// TIA Portal V17 export
// export: Created 2023-12-22T15:28:29.4431312Z, ExportSetting WithDefaults, DisplayName Totally Integrated Automation Portal, DisplayVersion V17, DisplayName TIA Portal Openness, DisplayVersion V17, DisplayName TIA Portal Version Control Interface, DisplayVersion V17, DisplayName STEP 7 Professional, DisplayVersion V17, DisplayName STEP 7 Safety, DisplayVersion V17, DisplayName WinCC Advanced, DisplayVersion V17
FUNCTION_BLOCK "Time_H"   // FB93, LAD
{ S7_Optimized_Access := 'FALSE' }
VERSION : 0.1
// stored: AutoNumber false, IsIECCheckEnabled false, SetENOAutomatically false, UDAEnableTagReadback false
   VAR DB_SPECIFIC
      SP_H { S7_SetPoint := 'True'} : DInt;   // Уставка часов - от 0 до 999
      SP_M { S7_SetPoint := 'True'} : DInt;   // Уставка минут - от 0 до 59
      SP_S { S7_SetPoint := 'True'} : DInt;   // Уставка секунд - от 0 до 59
      Now_H : DInt;   // Прошло часов от начала отсчёта
      Now_M : DInt;   // Прошло минут от начала отсчёта
      Now_S : DInt;   // Прошло секунд от начала отсчёта
      Rev_H : DInt;   // Осталось часов до уставки
      Rev_M : DInt;   // Осталось минут до уставки
      Rev_S : DInt;   // Осталось секунд до уставки
      Progress : Real;   // Прогресс выполнения
      Start : Bool;   // Запуск
      "Exit" : Bool;   // Счёт завершён
      Pause : Bool;   // Пауза
      Reset : Bool;   // Сброс таймера
   END_VAR
   VAR_TEMP
      Full_SP_S : DInt;
      Full_Now_S : DInt;
      Full_Delta_S : DInt;
      x1 : DInt;
      x2 : DInt;
   END_VAR
   VAR_TEMP   // added for the SCL form of the ladder/FBD networks
      _w1 : Bool;
      _w2 : Bool;
   END_VAR
BEGIN

REGION Network 1: Подсчёт времени
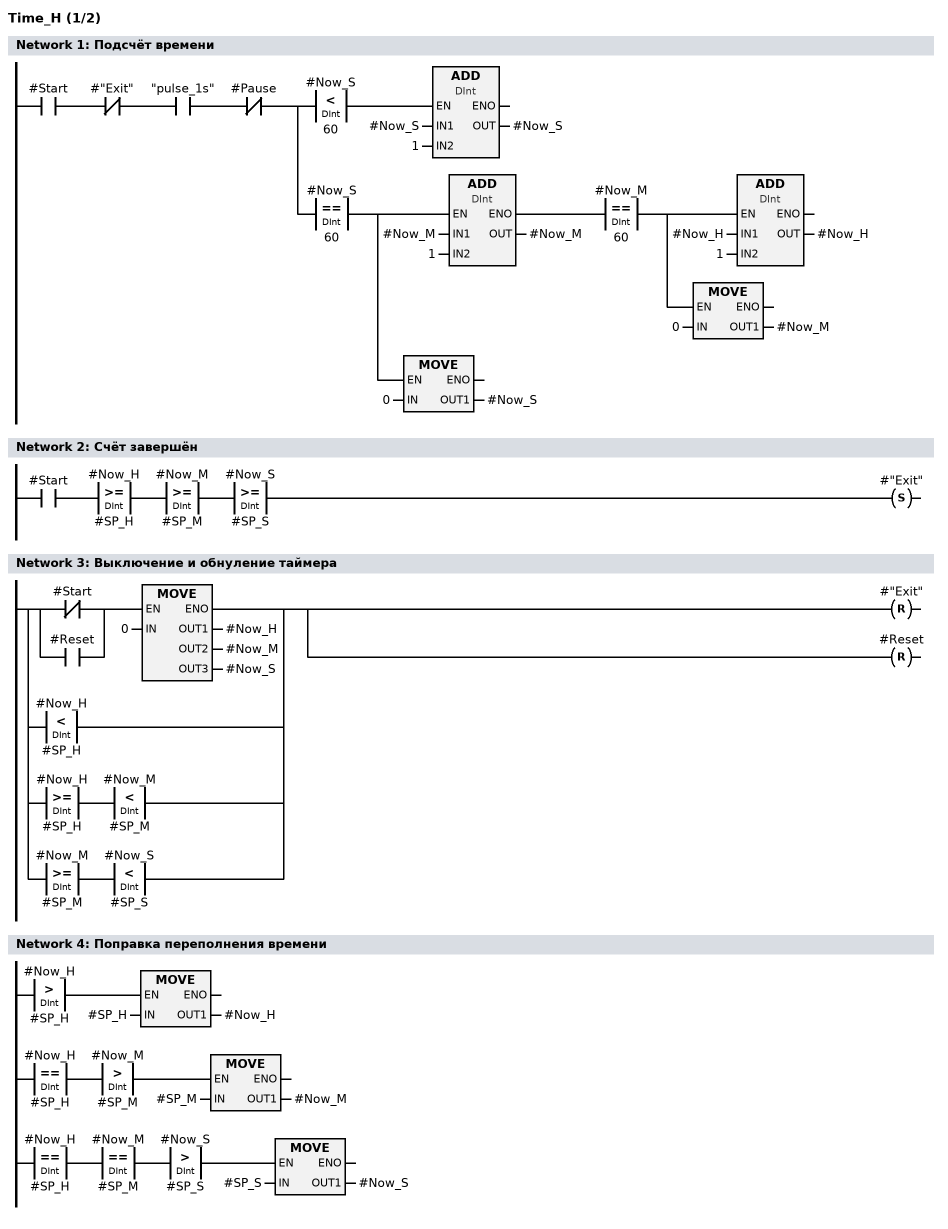
   RUNG wire#powerrail
      Contact( #Start )
      I_Contact( #"Exit" )
      Contact( "pulse_1s" )
      I_Contact( #Pause )
      wire#w1
      { S7_Templates := "SrcType := DInt" } LT_Contact(in1 := #Now_S, in2 := 60)
      { S7_Templates := "SrcType := DInt"; S7_GenerateENO := "TRUE" } Add(in1 := #Now_S, in2 := 1, out => #Now_S)
   END_RUNG
   RUNG wire#w1
      { S7_Templates := "SrcType := DInt" } EQ_Contact(in1 := #Now_S, in2 := 60)
      wire#w2
      { S7_Templates := "SrcType := DInt"; S7_GenerateENO := "TRUE" } Add(in1 := #Now_M, in2 := 1, out => #Now_M)
      { S7_Templates := "SrcType := DInt" } EQ_Contact(in1 := #Now_M, in2 := 60)
      wire#w3
      { S7_Templates := "SrcType := DInt"; S7_GenerateENO := "TRUE" } Add(in1 := #Now_H, in2 := 1, out => #Now_H)
   END_RUNG
   RUNG wire#w3
      { S7_GenerateENO := "TRUE" } Move(in := 0, out1 => #Now_M)
   END_RUNG
   RUNG wire#w2
      { S7_GenerateENO := "TRUE" } Move(in := 0, out1 => #Now_S)
   END_RUNG
   // the same network as SCL:
   // ENO of a box is taken as its EN; it also drops when the box reports an error
   #_w1 := #Start AND NOT #"Exit" AND "pulse_1s" AND NOT #Pause;
   IF #_w1 AND (#Now_S < 60) THEN #Now_S := #Now_S + 1; END_IF;
   #_w2 := #_w1 AND (#Now_S = 60);
   IF #_w2 THEN #Now_M := #Now_M + 1; END_IF;
   IF #_w2 AND (#Now_M = 60) THEN
       #Now_H := #Now_H + 1;
       #Now_M := 0;
   END_IF;
   IF #_w2 THEN #Now_S := 0; END_IF;
END_REGION

REGION Network 2: Счёт завершён
   RUNG wire#powerrail
      Contact( #Start )
      { S7_Templates := "SrcType := DInt" } GE_Contact(in1 := #Now_H, in2 := #SP_H)
      { S7_Templates := "SrcType := DInt" } GE_Contact(in1 := #Now_M, in2 := #SP_M)
      { S7_Templates := "SrcType := DInt" } GE_Contact(in1 := #Now_S, in2 := #SP_S)
      S_Coil( #"Exit" )
   END_RUNG
   // the same network as SCL:
   IF #Start AND (#Now_H >= #SP_H) AND (#Now_M >= #SP_M) AND (#Now_S >= #SP_S) THEN #"Exit" := TRUE; END_IF;
END_REGION

REGION Network 3: Выключение и обнуление таймера
   RUNG wire#powerrail
      I_Contact( #Start )
      wire#w1
      { S7_GenerateENO := "TRUE" } Move(in := 0, out1 => #Now_H, out2 => #Now_M, out3 => #Now_S)
      wire#w2
      R_Coil( #"Exit" )
   END_RUNG
   RUNG wire#powerrail
      Contact( #Reset )
   END_RUNG wire#w1
   RUNG wire#powerrail
      { S7_Templates := "SrcType := DInt" } LT_Contact(in1 := #Now_H, in2 := #SP_H)
   END_RUNG wire#w2
   RUNG wire#powerrail
      { S7_Templates := "SrcType := DInt" } GE_Contact(in1 := #Now_H, in2 := #SP_H)
      { S7_Templates := "SrcType := DInt" } LT_Contact(in1 := #Now_M, in2 := #SP_M)
   END_RUNG wire#w2
   RUNG wire#powerrail
      { S7_Templates := "SrcType := DInt" } GE_Contact(in1 := #Now_M, in2 := #SP_M)
      { S7_Templates := "SrcType := DInt" } LT_Contact(in1 := #Now_S, in2 := #SP_S)
   END_RUNG wire#w2
   RUNG wire#w2
      R_Coil( #Reset )
   END_RUNG
   // the same network as SCL:
   // ENO of a box is taken as its EN; it also drops when the box reports an error
   #_w1 := NOT #Start OR #Reset;
   IF #_w1 THEN
       #Now_H := 0;
       #Now_M := 0;
       #Now_S := 0;
   END_IF;
   IF #_w1 OR (#Now_H < #SP_H) OR ((#Now_H >= #SP_H) AND (#Now_M < #SP_M)) OR ((#Now_M >= #SP_M) AND (#Now_S < #SP_S)) THEN
       #"Exit" := FALSE;
       #Reset := FALSE;
   END_IF;
END_REGION

REGION Network 4: Поправка переполнения времени
   RUNG wire#powerrail
      { S7_Templates := "SrcType := DInt" } GT_Contact(in1 := #Now_H, in2 := #SP_H)
      { S7_GenerateENO := "TRUE" } Move(in := #SP_H, out1 => #Now_H)
   END_RUNG
   RUNG wire#powerrail
      { S7_Templates := "SrcType := DInt" } EQ_Contact(in1 := #Now_H, in2 := #SP_H)
      { S7_Templates := "SrcType := DInt" } GT_Contact(in1 := #Now_M, in2 := #SP_M)
      { S7_GenerateENO := "TRUE" } Move(in := #SP_M, out1 => #Now_M)
   END_RUNG
   RUNG wire#powerrail
      { S7_Templates := "SrcType := DInt" } EQ_Contact(in1 := #Now_H, in2 := #SP_H)
      { S7_Templates := "SrcType := DInt" } EQ_Contact(in1 := #Now_M, in2 := #SP_M)
      { S7_Templates := "SrcType := DInt" } GT_Contact(in1 := #Now_S, in2 := #SP_S)
      { S7_GenerateENO := "TRUE" } Move(in := #SP_S, out1 => #Now_S)
   END_RUNG
   // the same network as SCL:
   IF #Now_H > #SP_H THEN #Now_H := #SP_H; END_IF;
   IF (#Now_H = #SP_H) AND (#Now_M > #SP_M) THEN #Now_M := #SP_M; END_IF;
   IF (#Now_H = #SP_H) AND (#Now_M = #SP_M) AND (#Now_S > #SP_S) THEN #Now_S := #SP_S; END_IF;
END_REGION

REGION Network 5: Защита от некорретных значений
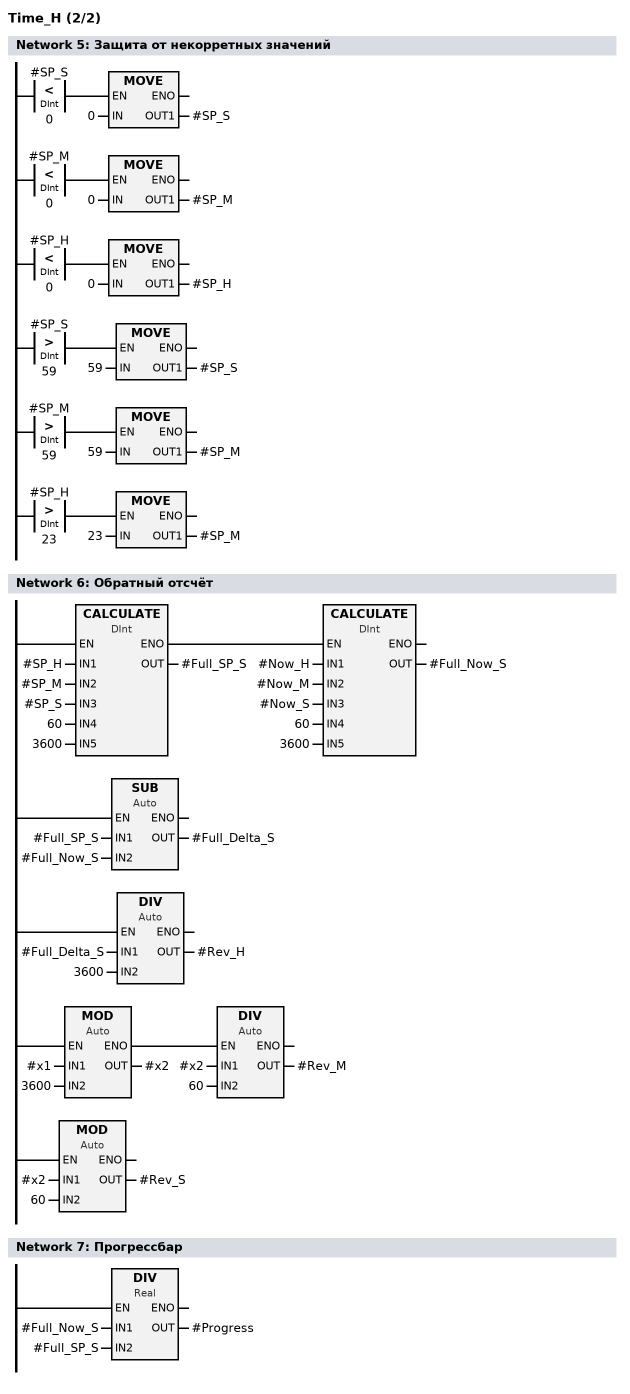
   RUNG wire#powerrail
      { S7_Templates := "SrcType := DInt" } LT_Contact(in1 := #SP_S, in2 := 0)
      { S7_GenerateENO := "TRUE" } Move(in := 0, out1 => #SP_S)
   END_RUNG
   RUNG wire#powerrail
      { S7_Templates := "SrcType := DInt" } LT_Contact(in1 := #SP_M, in2 := 0)
      { S7_GenerateENO := "TRUE" } Move(in := 0, out1 => #SP_M)
   END_RUNG
   RUNG wire#powerrail
      { S7_Templates := "SrcType := DInt" } LT_Contact(in1 := #SP_H, in2 := 0)
      { S7_GenerateENO := "TRUE" } Move(in := 0, out1 => #SP_H)
   END_RUNG
   RUNG wire#powerrail
      { S7_Templates := "SrcType := DInt" } GT_Contact(in1 := #SP_S, in2 := 59)
      { S7_GenerateENO := "TRUE" } Move(in := 59, out1 => #SP_S)
   END_RUNG
   RUNG wire#powerrail
      { S7_Templates := "SrcType := DInt" } GT_Contact(in1 := #SP_M, in2 := 59)
      { S7_GenerateENO := "TRUE" } Move(in := 59, out1 => #SP_M)
   END_RUNG
   RUNG wire#powerrail
      { S7_Templates := "SrcType := DInt" } GT_Contact(in1 := #SP_H, in2 := 23)
      { S7_GenerateENO := "TRUE" } Move(in := 23, out1 => #SP_M)
   END_RUNG
   // the same network as SCL:
   IF #SP_S < 0 THEN #SP_S := 0; END_IF;
   IF #SP_M < 0 THEN #SP_M := 0; END_IF;
   IF #SP_H < 0 THEN #SP_H := 0; END_IF;
   IF #SP_S > 59 THEN #SP_S := 59; END_IF;
   IF #SP_M > 59 THEN #SP_M := 59; END_IF;
   IF #SP_H > 23 THEN #SP_M := 23; END_IF;
END_REGION

REGION Network 6: Обратный отсчёт
   RUNG wire#powerrail
      { S7_Templates := "SrcType := DInt"; S7_Expression := "(IN1*IN4)+(IN2*IN5)+IN3" } Calculate(in1 := #SP_H, in2 := #SP_M, in3 := #SP_S, in4 := 60, in5 := 3600, out => #Full_SP_S)
      { S7_Templates := "SrcType := DInt"; S7_Expression := "(IN1*IN4)+(IN2*IN5)+IN3" } Calculate(in1 := #Now_H, in2 := #Now_M, in3 := #Now_S, in4 := 60, in5 := 3600, out => #Full_Now_S)
   END_RUNG
   RUNG wire#powerrail
      Sub(in1 := #Full_SP_S, in2 := #Full_Now_S, out => #Full_Delta_S)
   END_RUNG
   RUNG wire#powerrail
      Div(in1 := #Full_Delta_S, in2 := 3600, out => #Rev_H)
   END_RUNG
   RUNG wire#powerrail
      Mod(in1 := #x1, in2 := 3600, out => #x2)
      Div(in1 := #x2, in2 := 60, out => #Rev_M)
   END_RUNG
   RUNG wire#powerrail
      Mod(in1 := #x2, in2 := 60, out => #Rev_S)
   END_RUNG
   // the same network as SCL:
   #Full_SP_S := (#SP_H*60)+(#SP_M*3600)+#SP_S;
   #Full_Now_S := (#Now_H*60)+(#Now_M*3600)+#Now_S;
   #Full_Delta_S := #Full_SP_S - #Full_Now_S;
   #Rev_H := #Full_Delta_S / 3600;
   #x2 := #x1 MOD 3600;
   #Rev_M := #x2 / 60;
   #Rev_S := #x2 MOD 60;
END_REGION

REGION Network 7: Прогрессбар
   RUNG wire#powerrail
      { S7_Templates := "SrcType := Real" } Div(in1 := #Full_Now_S, in2 := #Full_SP_S, out => #Progress)
   END_RUNG
   // the same network as SCL:
   #Progress := #Full_Now_S / #Full_SP_S;
END_REGION
END_FUNCTION_BLOCK
